// TIA Portal V17 export
// export: Created 2026-07-18T05:18:21.7629844Z, ExportSetting WithDefaults, DisplayName Totally Integrated Automation Portal, DisplayVersion V17 Update 7, DisplayName TIA Portal Openness, DisplayVersion V17 Update 7, DisplayName TIA Portal Version Control Interface, DisplayVersion V17, DisplayName SINAMICS Startdrive Advanced, DisplayVersion V17 SP2, DisplayName SINAMICS Startdrive G110M, G120, G120C, G120D, G120P, G115D, DisplayVersion V17 SP2, DisplayName SINAMICS Startdrive G130, G150, S120, S150, SINAMICS MV, S210, DisplayVersion V17 SP2, DisplayName STEP 7 Professional, DisplayVersion V17 Update 7, DisplayName STEP 7 Safety, DisplayVersion V17 Update 6, DisplayName WinCC Advanced, DisplayVersion V17 Update 7
FUNCTION "FC_LAD_SimulateCylinder_Call" : Void   // FC1, LAD
{ S7_Optimized_Access := 'TRUE' }
VERSION : 0.1
// stored: AutoNumber true, IsIECCheckEnabled false, SetENOAutomatically false, UDAEnableTagReadback false
   VAR_INPUT
      btn_forward : Bool;
      btn_backward : Bool;
   END_VAR
   VAR_OUTPUT
      outputGoForwardPos : Bool;
      outputGoBackwardPos : Bool;
   END_VAR
   VAR_IN_OUT
      "io_Cylinder@ForwardPos" : Bool;
      "io_Cylinder@BackwardPos" : Bool;
   END_VAR
BEGIN

REGION Network 1
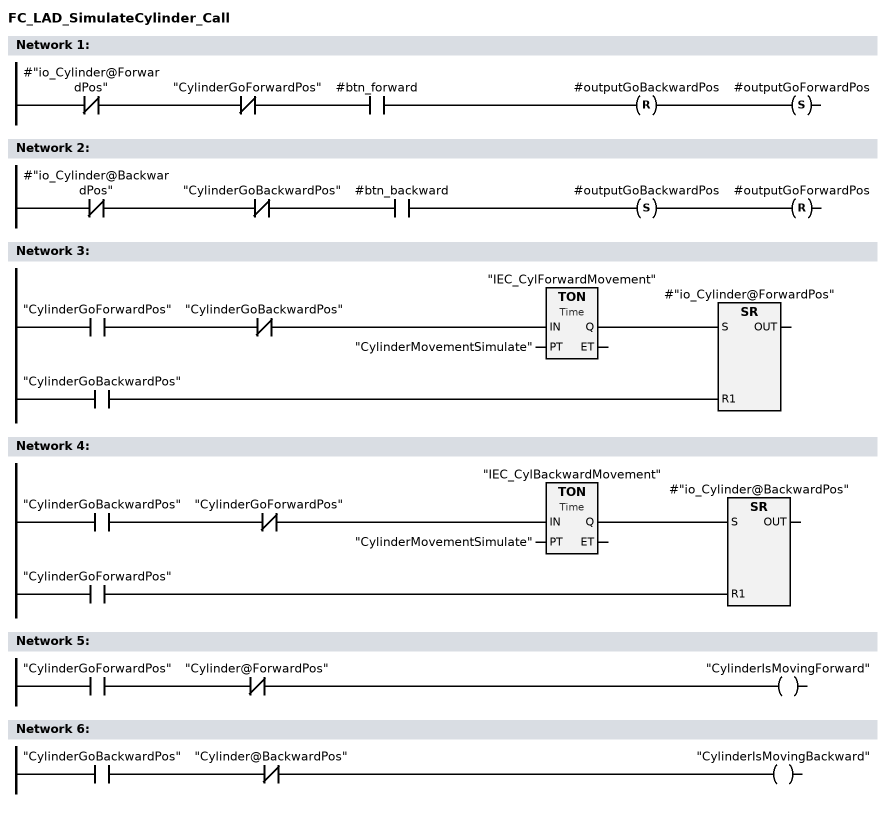
   RUNG wire#powerrail
      I_Contact( #"io_Cylinder@ForwardPos" )
      I_Contact( "CylinderGoForwardPos" )
      Contact( #btn_forward )
      R_Coil( #outputGoBackwardPos )
      S_Coil( #outputGoForwardPos )
   END_RUNG
   // the same network as SCL:
   IF NOT #"io_Cylinder@ForwardPos" AND NOT "CylinderGoForwardPos" AND #btn_forward THEN
       #outputGoBackwardPos := FALSE;
       #outputGoForwardPos := TRUE;
   END_IF;
END_REGION

REGION Network 2
   RUNG wire#powerrail
      I_Contact( #"io_Cylinder@BackwardPos" )
      I_Contact( "CylinderGoBackwardPos" )
      Contact( #btn_backward )
      S_Coil( #outputGoBackwardPos )
      R_Coil( #outputGoForwardPos )
   END_RUNG
   // the same network as SCL:
   IF NOT #"io_Cylinder@BackwardPos" AND NOT "CylinderGoBackwardPos" AND #btn_backward THEN
       #outputGoBackwardPos := TRUE;
       #outputGoForwardPos := FALSE;
   END_IF;
END_REGION

REGION Network 3
   RUNG wire#powerrail
      Contact( "CylinderGoForwardPos" )
      I_Contact( "CylinderGoBackwardPos" )
      { S7_Templates := "time_type := Time" } "IEC_CylForwardMovement".TON(pt := "CylinderMovementSimulate", et =>)
      S_SR(operand := #"io_Cylinder@ForwardPos", r1 := wire#w1)
   END_RUNG
   RUNG wire#powerrail
      Contact( "CylinderGoBackwardPos" )
   END_RUNG wire#w1
   // the same network as SCL:
   "IEC_CylForwardMovement".TON(IN := "CylinderGoForwardPos" AND NOT "CylinderGoBackwardPos",
                           PT := "CylinderMovementSimulate");
   IF "IEC_CylForwardMovement".Q THEN
       #"io_Cylinder@ForwardPos" := TRUE;   // SR flip-flop
   END_IF;
   IF "CylinderGoBackwardPos" THEN #"io_Cylinder@ForwardPos" := FALSE; END_IF;
END_REGION

REGION Network 4
   RUNG wire#powerrail
      Contact( "CylinderGoBackwardPos" )
      I_Contact( "CylinderGoForwardPos" )
      { S7_Templates := "time_type := Time" } "IEC_CylBackwardMovement".TON(pt := "CylinderMovementSimulate", et =>)
      S_SR(operand := #"io_Cylinder@BackwardPos", r1 := wire#w1)
   END_RUNG
   RUNG wire#powerrail
      Contact( "CylinderGoForwardPos" )
   END_RUNG wire#w1
   // the same network as SCL:
   "IEC_CylBackwardMovement".TON(IN := "CylinderGoBackwardPos" AND NOT "CylinderGoForwardPos",
                           PT := "CylinderMovementSimulate");
   IF "IEC_CylBackwardMovement".Q THEN
       #"io_Cylinder@BackwardPos" := TRUE;   // SR flip-flop
   END_IF;
   IF "CylinderGoForwardPos" THEN #"io_Cylinder@BackwardPos" := FALSE; END_IF;
END_REGION

REGION Network 5
   RUNG wire#powerrail
      Contact( "CylinderGoForwardPos" )
      I_Contact( "Cylinder@ForwardPos" )
      Coil( "CylinderIsMovingForward" )
   END_RUNG
   // the same network as SCL:
   "CylinderIsMovingForward" := "CylinderGoForwardPos" AND NOT "Cylinder@ForwardPos";
END_REGION

REGION Network 6
   RUNG wire#powerrail
      Contact( "CylinderGoBackwardPos" )
      I_Contact( "Cylinder@BackwardPos" )
      Coil( "CylinderIsMovingBackward" )
   END_RUNG
   // the same network as SCL:
   "CylinderIsMovingBackward" := "CylinderGoBackwardPos" AND NOT "Cylinder@BackwardPos";
END_REGION
END_FUNCTION
